Omron CX-Programmer project НовыйПроект (CX-Programmer 9.54)

# PLC НовыйПЛК1: CP1L-E EM

## Global symbols (name address type ; comment)
0.02 BOOL  ; EMG
0.08 BOOL  ; пустой латок
100.06 BOOL  ; лампа зеленой кнопки
C0000 BOOL  ; Счетчик шага ленты
C0001 BOOL  ; Счетчик часов
C0002 BOOL  ; Счетчик секунд
C0003 BOOL  ; Счетчик минут
C0004 BOOL  ; Счетчик счетчиков часов
C0005 BOOL  ; Счетчик ручного режима
C0006 BOOL  ; Счетчик аварий элеватора
C0007 BOOL  ; Счетчик аварий тарелки
C0008 BOOL  ; Счетчик нажатий грибка
C0009 BOOL  ; Счетчик реле безопасности
C0010 BOOL  ; счетсик секунд
C0011 BOOL  ; счетчик минут
C0012 BOOL  ; счтечик часов
C0013 BOOL  ; счетчик счетчика часов
C0014 BOOL  ; счетчик секунд
C0015 BOOL  ; счетчик минут
C0016 BOOL  ; счетчик часов
T0000 BOOL  ; Таймер задержки ленты
T0001 BOOL  ; лента не двигается
T0002 BOOL  ; Задержка включения ориентатора
T0005 BOOL  ; Задержка включения воздуха
T0006 BOOL  ; Задержка выключения ориентатора
T0010 BOOL  ; Наполнение тарелки
T0012 BOOL  ; лента не двигается
W0.03 BOOL  ; Ошибка связи с ПЧ
W0.04 BOOL  ; Связь с ПЧ ОК
W10.03 BOOL  ; Движение ленты с панели
W10.04 BOOL  ; Сброс
W1.01 BOOL  ; Ручная подача воздуха в трубу
W1.02 BOOL  ; Подача воздуха с панели
W1.09 BOOL  ; Сменился день
W2.01 BOOL  ; Общий сброс
W3.00 BOOL  ; сброс веремя работы
DayNew D600 UINT  ; Новый день
DayStar D602 UINT  ; День прошедший
LocAlarm D554 UINT
LocEMG D562 UINT
LocElev D558 UINT
LocManual D556 UINT
LocNotaus D564 UINT
LocTarelki D560 UINT
ResAlarm D504 UINT
ResEMG D512 UINT
ResElev D508 UINT
ResManual D506 UINT
ResNotaus D514 UINT
ResProst D500 UDINT  ; Простой после сброса
ResTarelki D510 UINT
ResWork D502 UDINT  ; Работа после сброса
Safety 0.00 BOOL  ; Реле безопасности
StatAlarm D464 UINT
StatEMG D468 UINT
StatElev D466 UINT
StatManual D465 UINT
StatNotaus D469 UINT
StatProst D460 UDINT  ; Глобальная статистика простоя
StatTarelki D467 UINT
StatWork D462 UDINT  ; Глобальная статистика работы
TimeSek A351 UINT
ghr INV002_Refresh_X31_
locProst D550 UDINT_BCD  ; время простоя локальное
locWork D552 UDINT_BCD  ; время работы локальное
time D400 UINT
Контроль_нового_дня Новый_день
Сброс_EMG Сброс2
Сброс_Ручного_режима Сброс2
Сброс_аварии_ленты Сброс2
Сброс_аварии_тарелки Сброс2
Сброс_аварии_терелки Сброс2
Сброс_времени_аварии Сброс2
Сброс_времени_работы Сброс
Сброс_реле_безопасности Сброс2
Смещение_EMG Сдвиг_данных2
Смещение_авари Сдвиг_данных2
Смещение_простоя сдвиг_данных
Смещение_работы сдвиг_данных
Смещение_реле_безопасности Сдвиг_данных2
Смещение_ручного Сдвиг_данных2
Смещение_тарелки Сдвиг_данных2
Смещение_элеватора Сдвиг_данных2
сброс_времени_простоя Сброс

## Program Ориентатор (cyclic task 0)
Local symbols
Air 100.00 BOOL  ; Подача воздуха
AirPipe 101.00 BOOL  ; Клапан воздуха в трубе
Alarm W0.02 BOOL  ; Сигнал ошибки
Alarm_Elevator W0.08 BOOL  ; Авария ленты
Alarm_Feeder W0.11 BOOL  ; Авария вращения тарелки
B1 0.04 BOOL  ; Заполнение тарелки
B2 0.03 BOOL  ; Уровень бункера
B3 0.06 BOOL  ; Шаг ленты
B4 0.05 BOOL  ; Вращение тарелки
B5 0.07 BOOL  ; Максимум лотка
DD434 INT
Flag W0.00 BOOL  ; Флаг старта
Freq D0 UINT  ; Задание частоты с панели
Green_Light 100.07 BOOL  ; Светофор зеленый
Manual W10.02 BOOL  ; Ручной режим
Power_Elevator 101.02 BOOL  ; Двигатель ленты
Power_Feeder W0.01 BOOL  ; Включение вращения тарелки
Red_Lamp 100.02 BOOL  ; Питание Реле
Red_Light 100.03 BOOL  ; Светофор красный
Reset W10.01 BOOL  ; Сброс
ResetSafety 100.01 BOOL  ; Сброс реле безопасности
Safety 0.00 BOOL  ; Реле безопасности
Sound 100.05 BOOL  ; Звук
Start W10.00 BOOL  ; Старт
Step D401 UINT_BCD  ; Количество шагов ленты
Timer1 D402 UINT_BCD  ; Задержка ленты
Timer2 D404 UINT_BCD  ; Задержка включения ориентатора
Timer3 D406 UINT_BCD  ; Задержка выключения ориентатора
Timer4 D408 UINT_BCD  ; Задержка подачи воздуха в трубе
Timer5 D410 UINT_BCD  ; Задержка отключения воздуха в трубе
Yellow_Light 100.04 BOOL  ; Светофор желтый
В431 CHANNEL
С13 INT

### Section Основная_программа

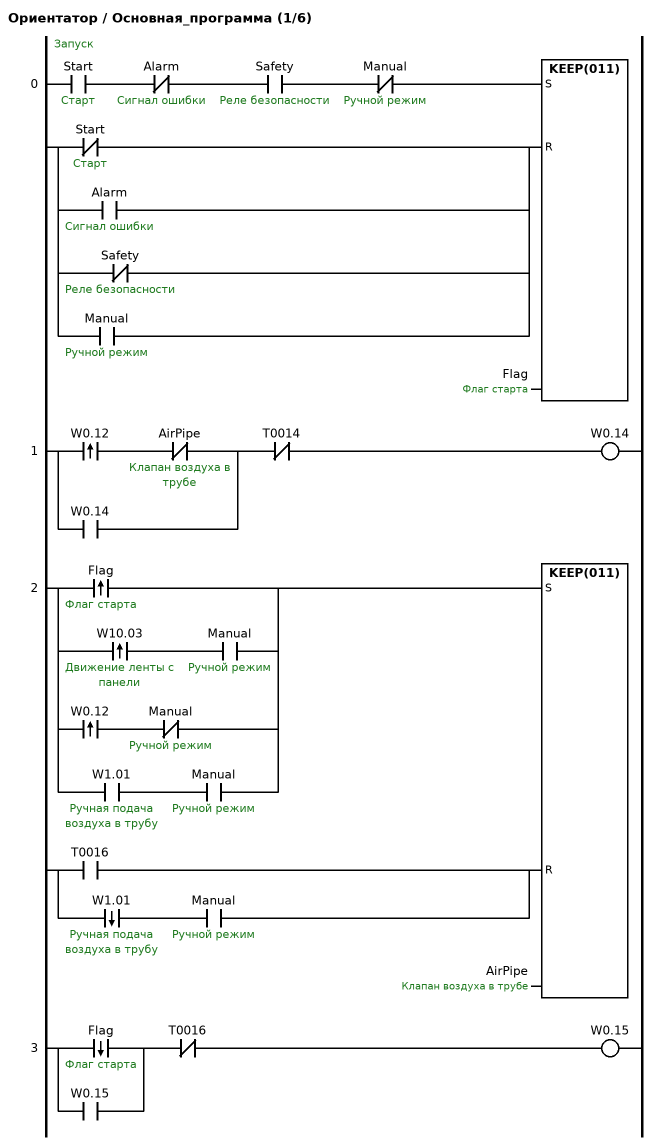
; rung 0: Запуск
LD Start  ; Старт
ANDNOT Alarm  ; Сигнал ошибки
AND Safety  ; Реле безопасности
ANDNOT Manual  ; Ручной режим
LDNOT Start  ; Старт
OR Alarm  ; Сигнал ошибки
ORNOT Safety  ; Реле безопасности
OR Manual  ; Ручной режим
KEEP(011) Flag  ; Флаг старта
; rung 1
@LD W0.12
ANDNOT AirPipe  ; Клапан воздуха в трубе
OR W0.14
ANDNOT T0014
OUT W0.14
; rung 2
@LD Flag  ; Флаг старта
@LD W10.03  ; Движение ленты с панели
AND Manual  ; Ручной режим
ORLD
@LD W0.12
ANDNOT Manual  ; Ручной режим
ORLD
LD W1.01  ; Ручная подача воздуха в трубу
AND Manual  ; Ручной режим
ORLD
LD T0016
%LD W1.01  ; Ручная подача воздуха в трубу
AND Manual  ; Ручной режим
ORLD
KEEP(011) AirPipe  ; Клапан воздуха в трубе
; rung 3
%LD Flag  ; Флаг старта
OR W0.15
ANDNOT T0016
OUT W0.15

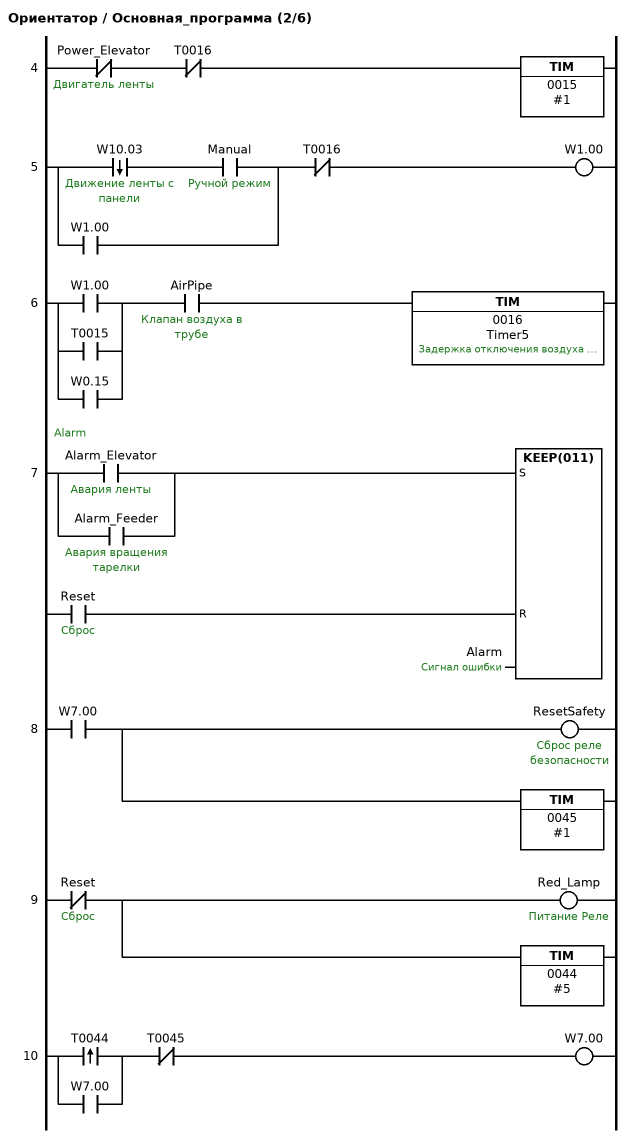
; rung 4
LDNOT Power_Elevator  ; Двигатель ленты
ANDNOT T0016
TIM 0015 #1
; rung 5
%LD W10.03  ; Движение ленты с панели
AND Manual  ; Ручной режим
OR W1.00
ANDNOT T0016
OUT W1.00
; rung 6
LD W1.00
OR T0015
OR W0.15
AND AirPipe  ; Клапан воздуха в трубе
TIM 0016 Timer5  ; Задержка отключения воздуха в трубе
; rung 7: Alarm
LD Alarm_Elevator  ; Авария ленты
OR Alarm_Feeder  ; Авария вращения тарелки
LD Reset  ; Сброс
KEEP(011) Alarm  ; Сигнал ошибки
; rung 8
LD W7.00
OUT ResetSafety  ; Сброс реле безопасности
TIM 0045 #1
; rung 9
LDNOT Reset  ; Сброс
OUT Red_Lamp  ; Питание Реле
TIM 0044 #5
; rung 10
@LD T0044
OR W7.00
ANDNOT T0045
OUT W7.00

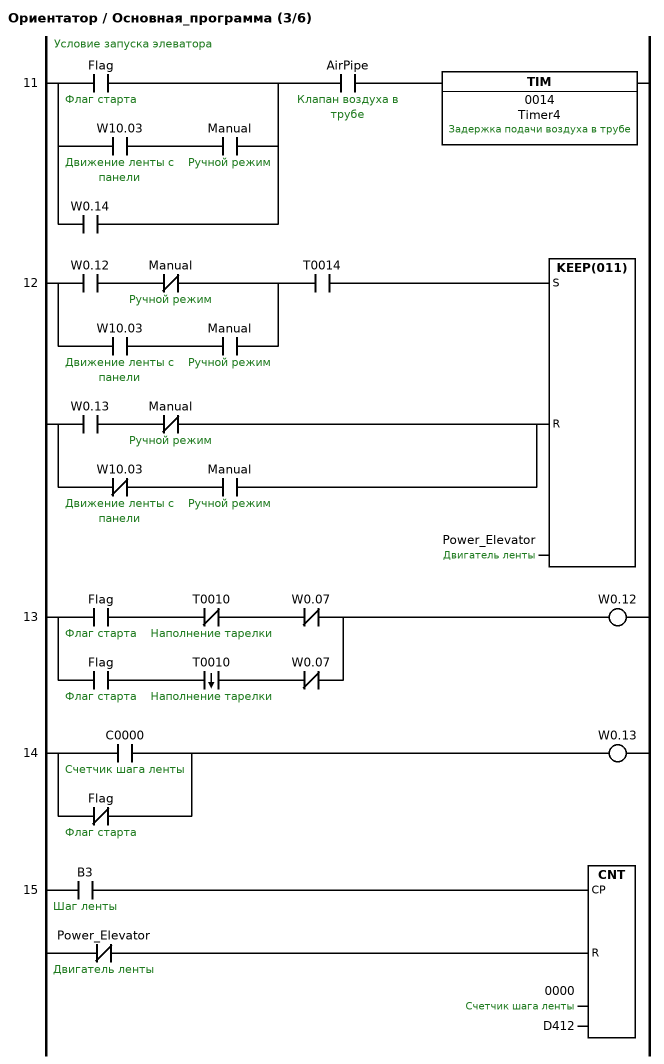
; rung 11: Условие запуска элеватора
LD Flag  ; Флаг старта
LD W10.03  ; Движение ленты с панели
AND Manual  ; Ручной режим
ORLD
OR W0.14
AND AirPipe  ; Клапан воздуха в трубе
TIM 0014 Timer4  ; Задержка подачи воздуха в трубе
; rung 12
LD W0.12
ANDNOT Manual  ; Ручной режим
LD W10.03  ; Движение ленты с панели
AND Manual  ; Ручной режим
ORLD
AND T0014
LD W0.13
ANDNOT Manual  ; Ручной режим
LDNOT W10.03  ; Движение ленты с панели
AND Manual  ; Ручной режим
ORLD
KEEP(011) Power_Elevator  ; Двигатель ленты
; rung 13
LD Flag  ; Флаг старта
ANDNOT T0010  ; Наполнение тарелки
ANDNOT W0.07
LD Flag  ; Флаг старта
%AND T0010  ; Наполнение тарелки
ANDNOT W0.07
ORLD
OUT W0.12
; rung 14
LD C0000  ; Счетчик шага ленты
ORNOT Flag  ; Флаг старта
OUT W0.13
; rung 15
LD B3  ; Шаг ленты
LDNOT Power_Elevator  ; Двигатель ленты
CNT 0000 D412  ; Счетчик шага ленты

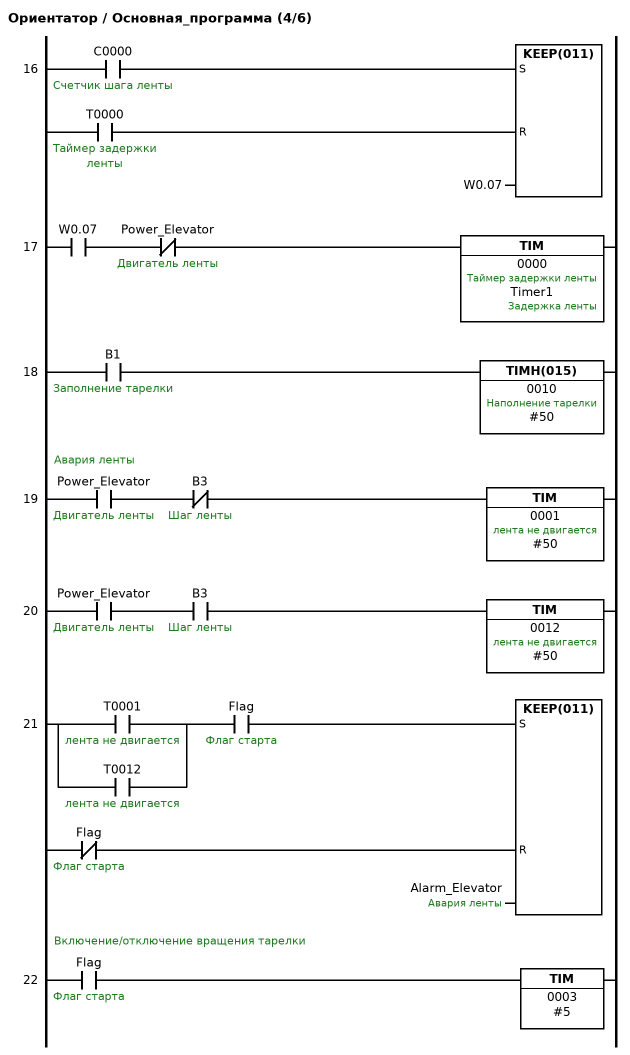
; rung 16
LD C0000  ; Счетчик шага ленты
LD T0000  ; Таймер задержки ленты
KEEP(011) W0.07
; rung 17
LD W0.07
ANDNOT Power_Elevator  ; Двигатель ленты
TIM 0000 Timer1  ; Задержка ленты, Таймер задержки ленты
; rung 18
LD B1  ; Заполнение тарелки
TIMH(015) 0010 #50  ; Наполнение тарелки
; rung 19: Авария ленты
LD Power_Elevator  ; Двигатель ленты
ANDNOT B3  ; Шаг ленты
TIM 0001 #50  ; лента не двигается
; rung 20
LD Power_Elevator  ; Двигатель ленты
AND B3  ; Шаг ленты
TIM 0012 #50  ; лента не двигается
; rung 21
LD T0001  ; лента не двигается
OR T0012  ; лента не двигается
AND Flag  ; Флаг старта
LDNOT Flag  ; Флаг старта
KEEP(011) Alarm_Elevator  ; Авария ленты
; rung 22: Включение/отключение вращения тарелки
LD Flag  ; Флаг старта
TIM 0003 #5

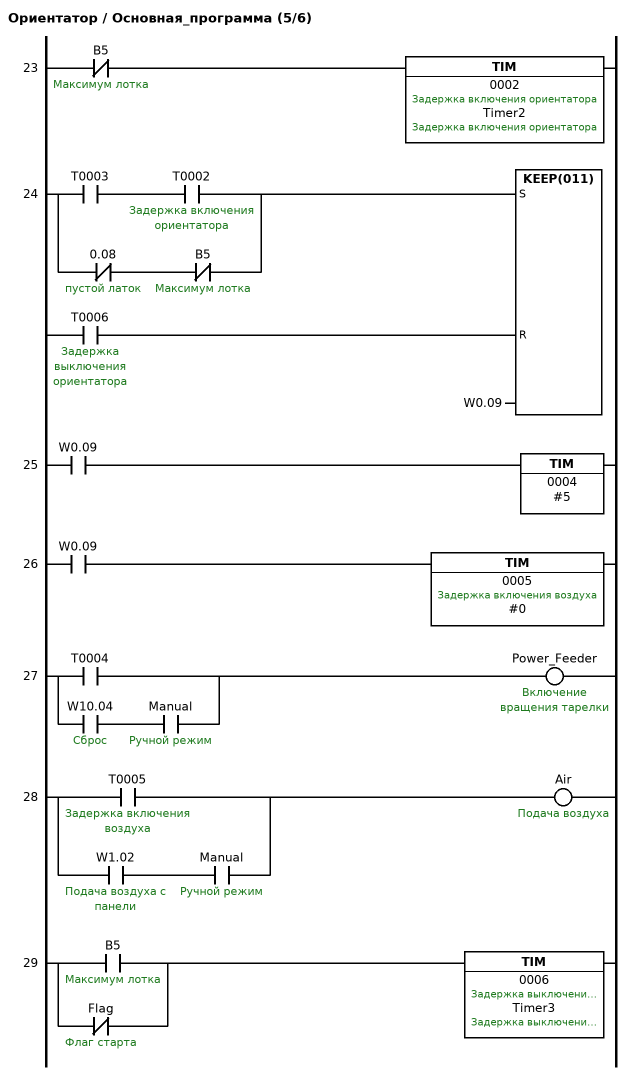
; rung 23
LDNOT B5  ; Максимум лотка
TIM 0002 Timer2  ; Задержка включения ориентатора
; rung 24
LD T0003
AND T0002  ; Задержка включения ориентатора
LDNOT 0.08  ; пустой латок
ANDNOT B5  ; Максимум лотка
ORLD
LD T0006  ; Задержка выключения ориентатора
KEEP(011) W0.09
; rung 25
LD W0.09
TIM 0004 #5
; rung 26
LD W0.09
TIM 0005 #0  ; Задержка включения воздуха
; rung 27
LD T0004
LD W10.04  ; Сброс
AND Manual  ; Ручной режим
ORLD
OUT Power_Feeder  ; Включение вращения тарелки
; rung 28
LD T0005  ; Задержка включения воздуха
LD W1.02  ; Подача воздуха с панели
AND Manual  ; Ручной режим
ORLD
OUT Air  ; Подача воздуха
; rung 29
LD B5  ; Максимум лотка
ORNOT Flag  ; Флаг старта
TIM 0006 Timer3  ; Задержка выключения ориентатора

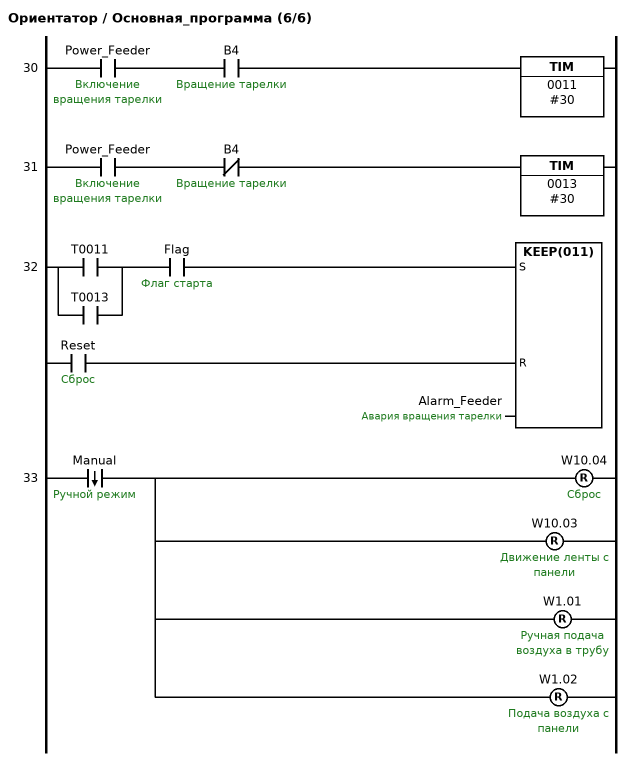
; rung 30
LD Power_Feeder  ; Включение вращения тарелки
AND B4  ; Вращение тарелки
TIM 0011 #30
; rung 31
LD Power_Feeder  ; Включение вращения тарелки
ANDNOT B4  ; Вращение тарелки
TIM 0013 #30
; rung 32
LD T0011
OR T0013
AND Flag  ; Флаг старта
LD Reset  ; Сброс
KEEP(011) Alarm_Feeder  ; Авария вращения тарелки
; rung 33
%LD Manual  ; Ручной режим
RSET W10.04  ; Сброс
RSET W10.03  ; Движение ленты с панели
RSET W1.01  ; Ручная подача воздуха в трубу
RSET W1.02  ; Подача воздуха с панели

### Section Частотник

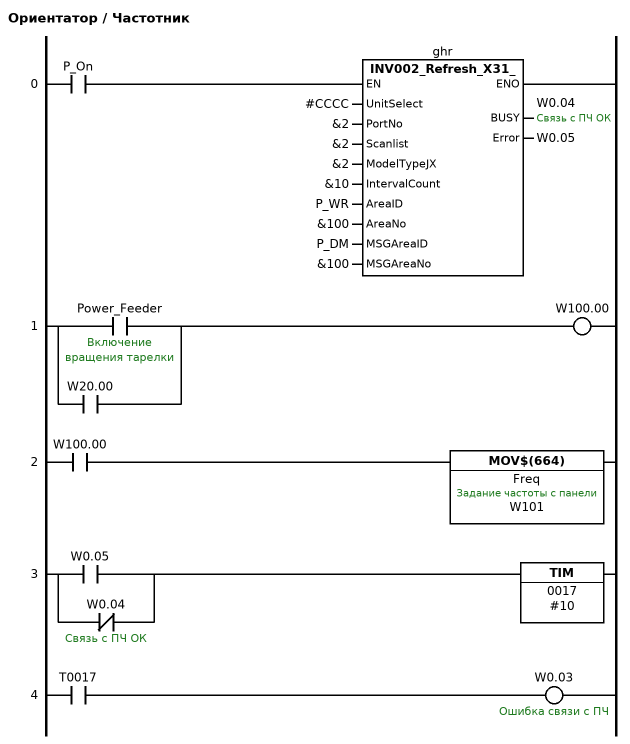
; rung 0
LD P_On
CALL ghr : INV002_Refresh_X31_ (UnitSelect := #CCCC, PortNo := &2, Scanlist := &2, ModelTypeJX := &2, IntervalCount := &10, AreaID := P_WR, AreaNo := &100, MSGAreaID := P_DM, MSGAreaNo := &100, BUSY => W0.04, Error => W0.05)  ; Связь с ПЧ ОК
; rung 1
LD Power_Feeder  ; Включение вращения тарелки
OR W20.00
OUT W100.00
; rung 2
LD W100.00
MOV$(664) Freq W101  ; Задание частоты с панели
; rung 3
LD W0.05
ORNOT W0.04  ; Связь с ПЧ ОК
TIM 0017 #10
; rung 4
LD T0017
OUT W0.03  ; Ошибка связи с ПЧ

### Section Индикация

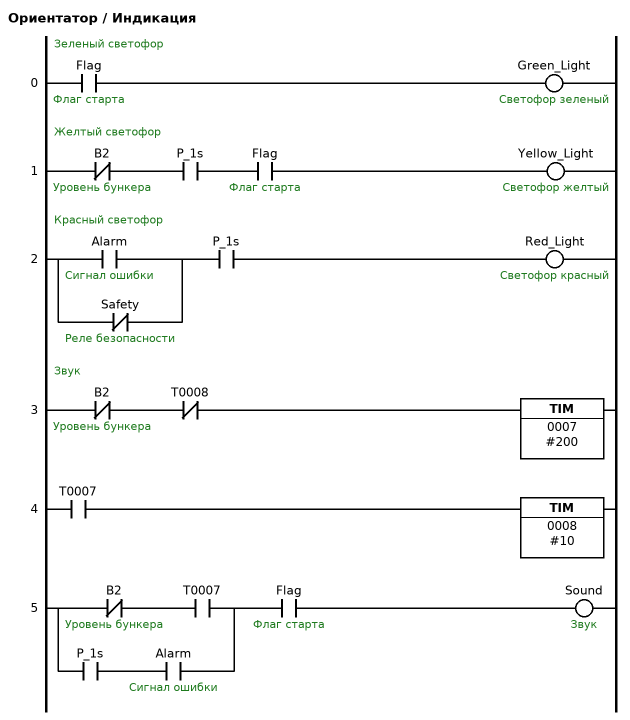
; rung 0: Зеленый светофор
LD Flag  ; Флаг старта
OUT Green_Light  ; Светофор зеленый
; rung 1: Желтый светофор
LDNOT B2  ; Уровень бункера
AND P_1s
AND Flag  ; Флаг старта
OUT Yellow_Light  ; Светофор желтый
; rung 2: Красный светофор
LD Alarm  ; Сигнал ошибки
ORNOT Safety  ; Реле безопасности
AND P_1s
OUT Red_Light  ; Светофор красный
; rung 3: Звук
LDNOT B2  ; Уровень бункера
ANDNOT T0008
TIM 0007 #200
; rung 4
LD T0007
TIM 0008 #10
; rung 5
LDNOT B2  ; Уровень бункера
AND T0007
LD P_1s
AND Alarm  ; Сигнал ошибки
ORLD
AND Flag  ; Флаг старта
OUT Sound  ; Звук

### Section End
; rung 0
END(001)

## Program статистика (cyclic task 1)
Local symbols
Alarm W0.02 BOOL  ; Сигнал ошибки
AlarmDay1 D628 UINT
AlarmDay2 D629 UINT
AlarmDay3 D630 UINT
Alarm_Elevator W0.08 BOOL  ; Авария ленты
Alarm_Feeder W0.11 BOOL  ; Авария вращения тарелки
Day1 D613 UINT
Day2 D616 UINT
Day3 D619 UINT
DayNew D600 UINT
DayStar D602 UINT
EMGDay1 D644 UINT
EMGDay2 D645 UINT
EMGDay3 D646 UINT
ElevDay1 D636 UINT
ElevDay2 D637 UINT
ElevDay3 D638 UINT
Flag W0.00 BOOL  ; Флаг старта
LocProst D550 UDINT
LocWork D552 UDINT
Manual W10.02 BOOL  ; Ручной режим
ManualDay1 D632 UINT
ManualDay2 D633 UINT
ManualDay3 D634 UINT
Mon1 D614 UINT
Mon2 D617 UINT
Mon3 D620 UINT
MonNew D601 UINT
MonStar D603 UINT
NotausDay1 D648 UINT
NotausDay2 D649 UINT
NotausDay3 D650 UINT
ProstDay1 D612 UINT  ; Простой 1 день
ProstDay2 D615 UINT  ; Простой 2 день
ProstDay3 D618 UINT  ; Простой 3 день
TarelkaDay1 D640 UINT
TarelkaDay2 D641 UINT
TarelkaDay3 D642 UINT
TochOtschAlarm D626 UINT
TochOtschEMG D643 UINT
TochOtschElev D635 UINT
TochOtschManual D631 UINT
TochOtschNotaus D647 UINT
TochOtschProst D610 UDINT
TochOtschTarelki D639 UINT
TochOtschWork D621 UDINT
WorkDay1 D623 UINT  ; работа 1 дня
WorkDay2 D624 UINT  ; Работа 2 дня
WorkDay3 D625 UINT  ; Работа 3 дня

### Section Сбор_статистики

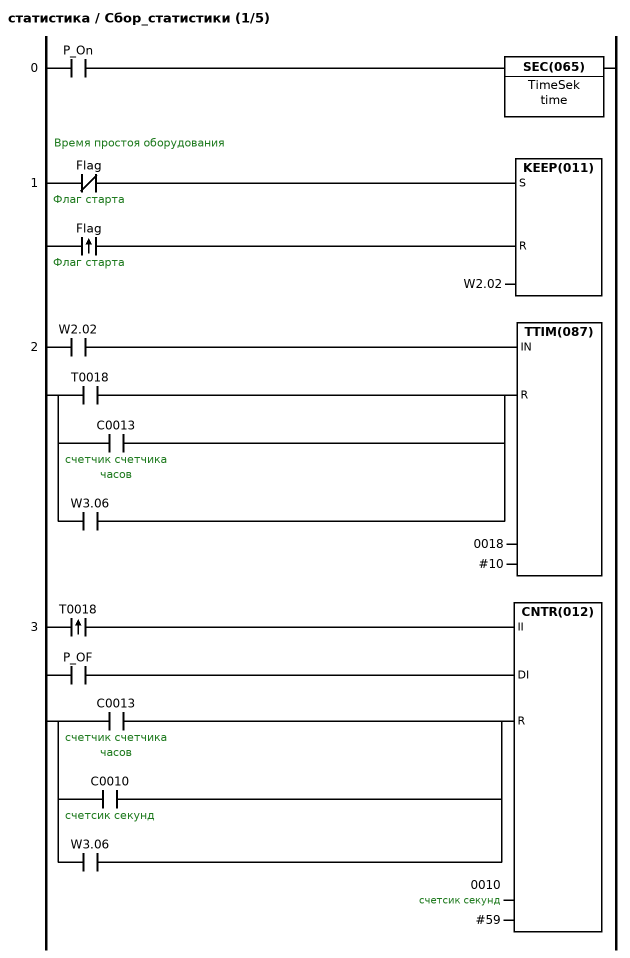
; rung 0
LD P_On
SEC(065) TimeSek time
; rung 1: Время простоя оборудования
LDNOT Flag  ; Флаг старта
@LD Flag  ; Флаг старта
KEEP(011) W2.02
; rung 2
LD W2.02
LD T0018
OR C0013  ; счетчик счетчика часов
OR W3.06
TTIM(087) 0018 #10
; rung 3
@LD T0018
LD P_OF
LD C0013  ; счетчик счетчика часов
OR C0010  ; счетсик секунд
OR W3.06
CNTR(012) 0010 #59  ; счетсик секунд

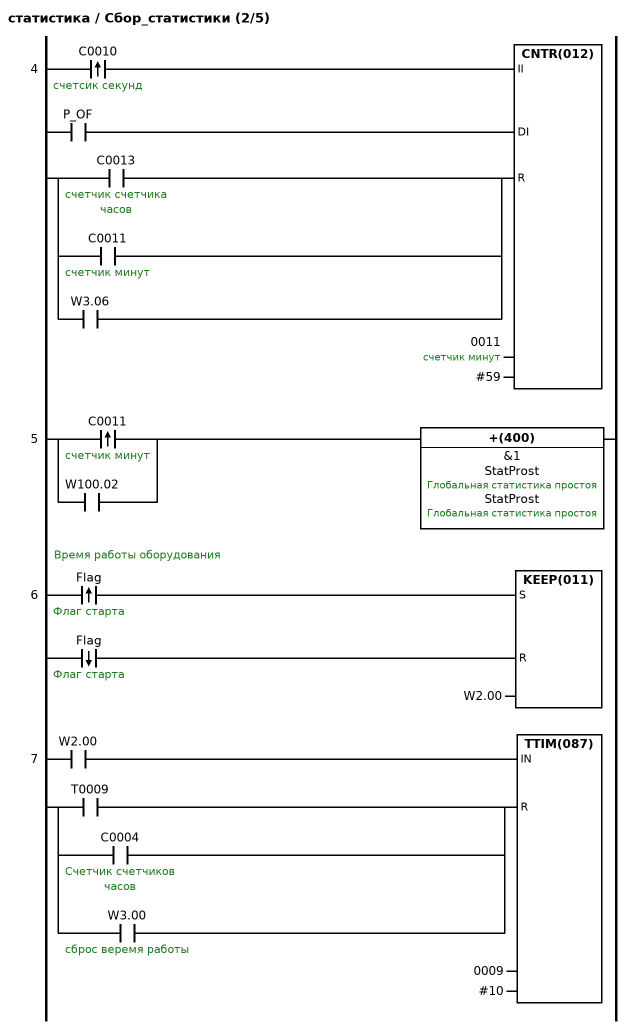
; rung 4
@LD C0010  ; счетсик секунд
LD P_OF
LD C0013  ; счетчик счетчика часов
OR C0011  ; счетчик минут
OR W3.06
CNTR(012) 0011 #59  ; счетчик минут
; rung 5
@LD C0011  ; счетчик минут
OR W100.02
+(400) &1 StatProst StatProst  ; Глобальная статистика простоя
; rung 6: Время работы оборудования
@LD Flag  ; Флаг старта
%LD Flag  ; Флаг старта
KEEP(011) W2.00
; rung 7
LD W2.00
LD T0009
OR C0004  ; Счетчик счетчиков часов
OR W3.00  ; сброс веремя работы
TTIM(087) 0009 #10

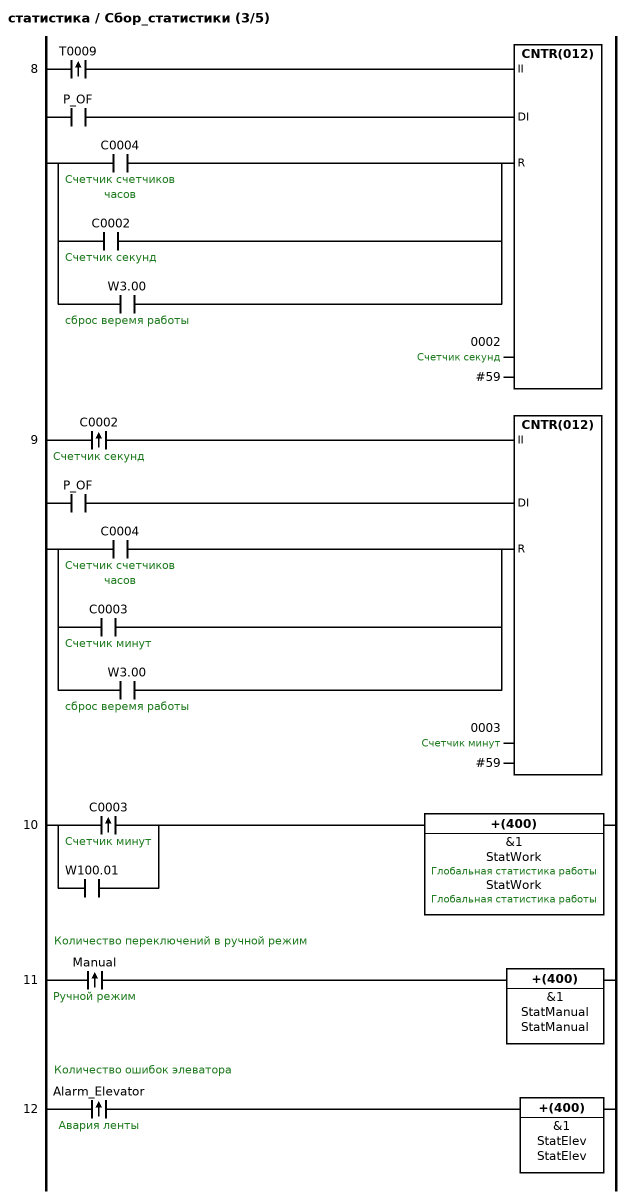
; rung 8
@LD T0009
LD P_OF
LD C0004  ; Счетчик счетчиков часов
OR C0002  ; Счетчик секунд
OR W3.00  ; сброс веремя работы
CNTR(012) 0002 #59  ; Счетчик секунд
; rung 9
@LD C0002  ; Счетчик секунд
LD P_OF
LD C0004  ; Счетчик счетчиков часов
OR C0003  ; Счетчик минут
OR W3.00  ; сброс веремя работы
CNTR(012) 0003 #59  ; Счетчик минут
; rung 10
@LD C0003  ; Счетчик минут
OR W100.01
+(400) &1 StatWork StatWork  ; Глобальная статистика работы
; rung 11: Количество переключений в ручной режим
@LD Manual  ; Ручной режим
+(400) &1 StatManual StatManual
; rung 12: Количество ошибок элеватора
@LD Alarm_Elevator  ; Авария ленты
+(400) &1 StatElev StatElev

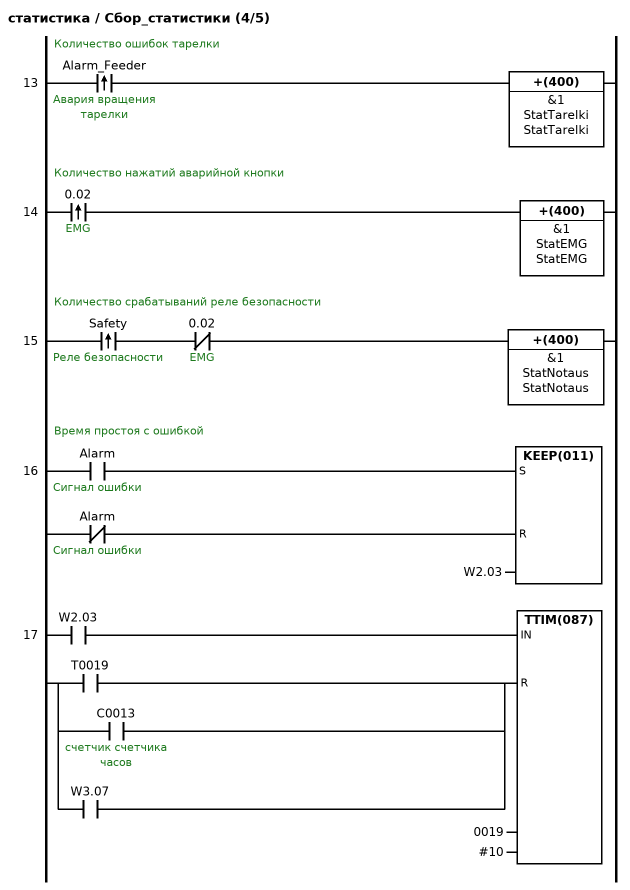
; rung 13: Количество ошибок тарелки
@LD Alarm_Feeder  ; Авария вращения тарелки
+(400) &1 StatTarelki StatTarelki
; rung 14: Количество нажатий аварийной кнопки
@LD 0.02  ; EMG
+(400) &1 StatEMG StatEMG
; rung 15: Количество срабатываний реле безопасности
@LD Safety  ; Реле безопасности
ANDNOT 0.02  ; EMG
+(400) &1 StatNotaus StatNotaus
; rung 16: Время простоя с ошибкой
LD Alarm  ; Сигнал ошибки
LDNOT Alarm  ; Сигнал ошибки
KEEP(011) W2.03
; rung 17
LD W2.03
LD T0019
OR C0013  ; счетчик счетчика часов
OR W3.07
TTIM(087) 0019 #10

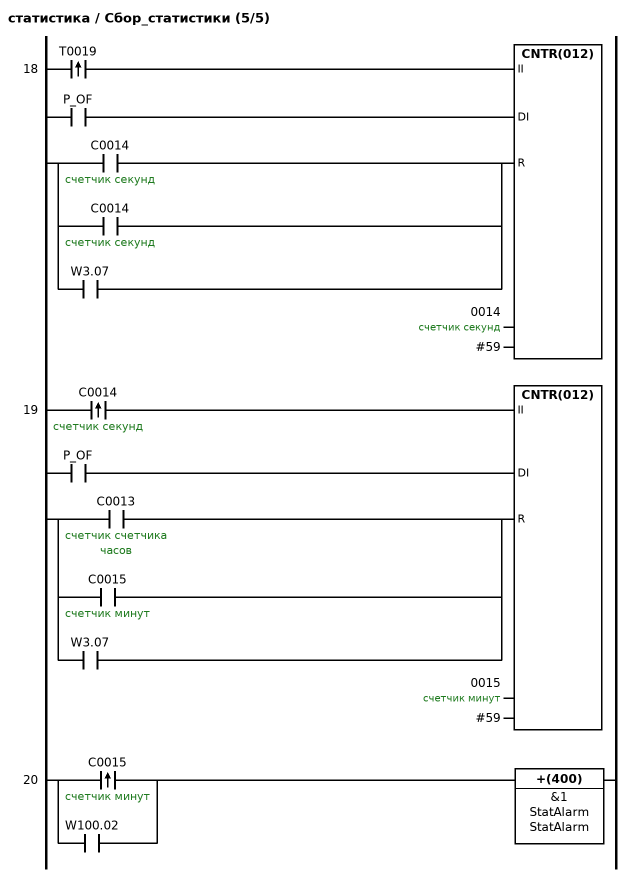
; rung 18
@LD T0019
LD P_OF
LD C0014  ; счетчик секунд
OR C0014  ; счетчик секунд
OR W3.07
CNTR(012) 0014 #59  ; счетчик секунд
; rung 19
@LD C0014  ; счетчик секунд
LD P_OF
LD C0013  ; счетчик счетчика часов
OR C0015  ; счетчик минут
OR W3.07
CNTR(012) 0015 #59  ; счетчик минут
; rung 20
@LD C0015  ; счетчик минут
OR W100.02
+(400) &1 StatAlarm StatAlarm

### Section расчет_статистики

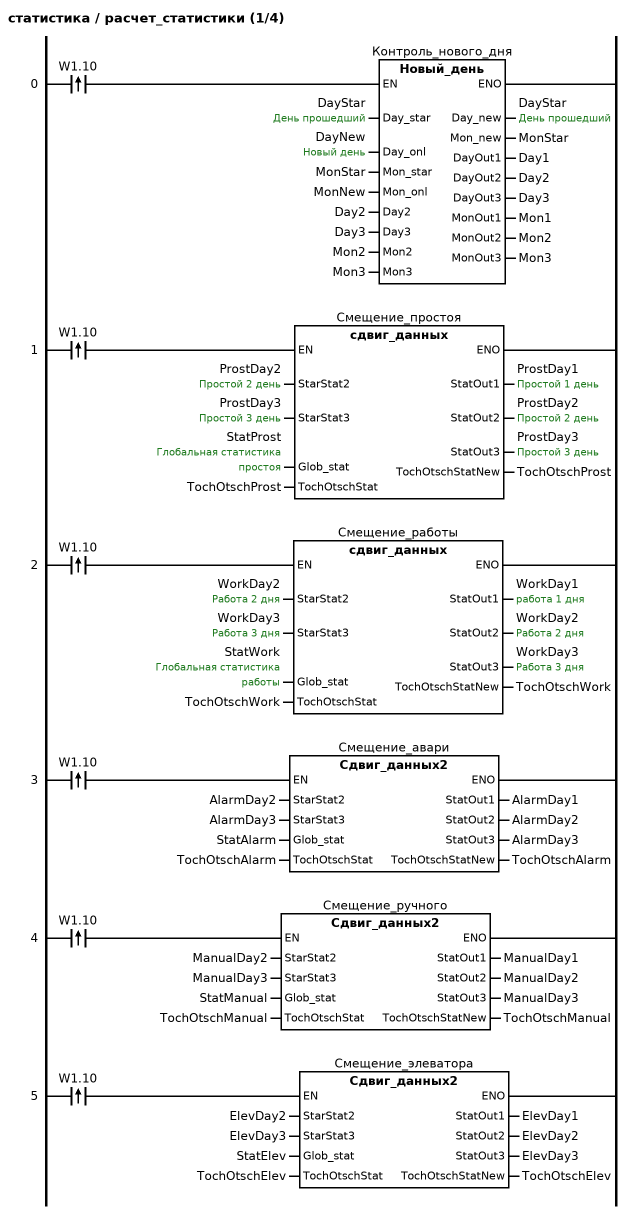
; rung 0
@LD W1.10
CALL Контроль_нового_дня : Новый_день (Day_star := DayStar, Day_onl := DayNew, Mon_star := MonStar, Mon_onl := MonNew, Day2 := Day2, Day3 := Day3, Mon2 := Mon2, Mon3 := Mon3, Day_new => DayStar, Mon_new => MonStar, DayOut1 => Day1, DayOut2 => Day2, DayOut3 => Day3, MonOut1 => Mon1, MonOut2 => Mon2, MonOut3 => Mon3)  ; День прошедший, Новый день
; rung 1
@LD W1.10
CALL Смещение_простоя : сдвиг_данных (StarStat2 := ProstDay2, StarStat3 := ProstDay3, Glob_stat := StatProst, TochOtschStat := TochOtschProst, StatOut1 => ProstDay1, StatOut2 => ProstDay2, StatOut3 => ProstDay3, TochOtschStatNew => TochOtschProst)  ; Простой 2 день, Простой 3 день, Глобальная статистика простоя, Простой 1 день
; rung 2
@LD W1.10
CALL Смещение_работы : сдвиг_данных (StarStat2 := WorkDay2, StarStat3 := WorkDay3, Glob_stat := StatWork, TochOtschStat := TochOtschWork, StatOut1 => WorkDay1, StatOut2 => WorkDay2, StatOut3 => WorkDay3, TochOtschStatNew => TochOtschWork)  ; Работа 2 дня, Работа 3 дня, Глобальная статистика работы, работа 1 дня
; rung 3
@LD W1.10
CALL Смещение_авари : Сдвиг_данных2 (StarStat2 := AlarmDay2, StarStat3 := AlarmDay3, Glob_stat := StatAlarm, TochOtschStat := TochOtschAlarm, StatOut1 => AlarmDay1, StatOut2 => AlarmDay2, StatOut3 => AlarmDay3, TochOtschStatNew => TochOtschAlarm)
; rung 4
@LD W1.10
CALL Смещение_ручного : Сдвиг_данных2 (StarStat2 := ManualDay2, StarStat3 := ManualDay3, Glob_stat := StatManual, TochOtschStat := TochOtschManual, StatOut1 => ManualDay1, StatOut2 => ManualDay2, StatOut3 => ManualDay3, TochOtschStatNew => TochOtschManual)
; rung 5
@LD W1.10
CALL Смещение_элеватора : Сдвиг_данных2 (StarStat2 := ElevDay2, StarStat3 := ElevDay3, Glob_stat := StatElev, TochOtschStat := TochOtschElev, StatOut1 => ElevDay1, StatOut2 => ElevDay2, StatOut3 => ElevDay3, TochOtschStatNew => TochOtschElev)

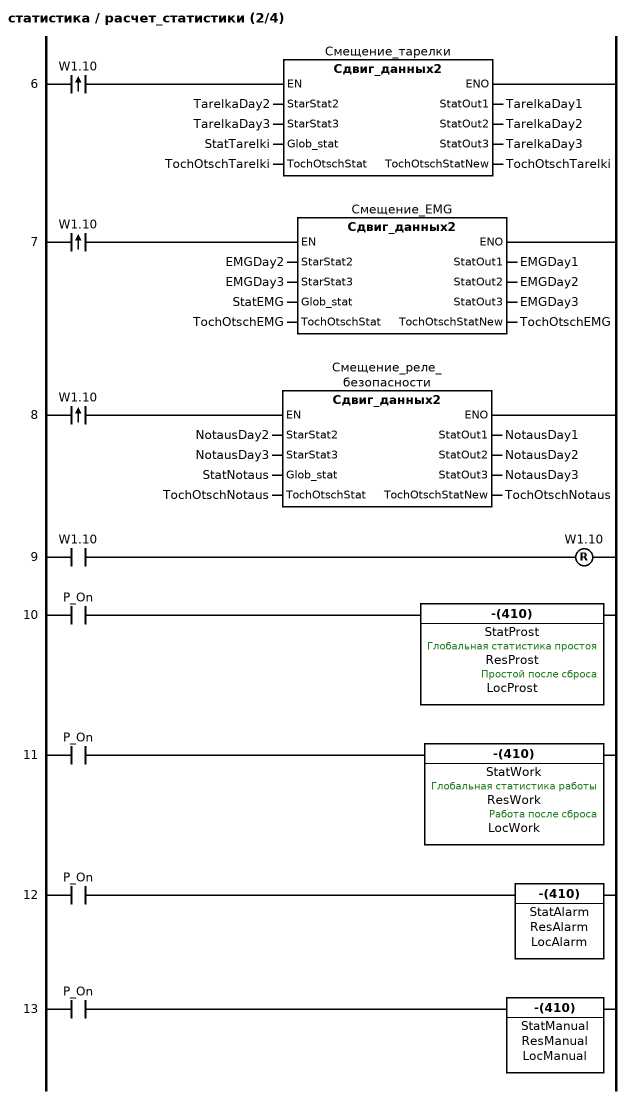
; rung 6
@LD W1.10
CALL Смещение_тарелки : Сдвиг_данных2 (StarStat2 := TarelkaDay2, StarStat3 := TarelkaDay3, Glob_stat := StatTarelki, TochOtschStat := TochOtschTarelki, StatOut1 => TarelkaDay1, StatOut2 => TarelkaDay2, StatOut3 => TarelkaDay3, TochOtschStatNew => TochOtschTarelki)
; rung 7
@LD W1.10
CALL Смещение_EMG : Сдвиг_данных2 (StarStat2 := EMGDay2, StarStat3 := EMGDay3, Glob_stat := StatEMG, TochOtschStat := TochOtschEMG, StatOut1 => EMGDay1, StatOut2 => EMGDay2, StatOut3 => EMGDay3, TochOtschStatNew => TochOtschEMG)
; rung 8
@LD W1.10
CALL Смещение_реле_безопасности : Сдвиг_данных2 (StarStat2 := NotausDay2, StarStat3 := NotausDay3, Glob_stat := StatNotaus, TochOtschStat := TochOtschNotaus, StatOut1 => NotausDay1, StatOut2 => NotausDay2, StatOut3 => NotausDay3, TochOtschStatNew => TochOtschNotaus)
; rung 9
LD W1.10
RSET W1.10
; rung 10
LD P_On
-(410) StatProst ResProst LocProst  ; Глобальная статистика простоя, Простой после сброса
; rung 11
LD P_On
-(410) StatWork ResWork LocWork  ; Глобальная статистика работы, Работа после сброса
; rung 12
LD P_On
-(410) StatAlarm ResAlarm LocAlarm
; rung 13
LD P_On
-(410) StatManual ResManual LocManual

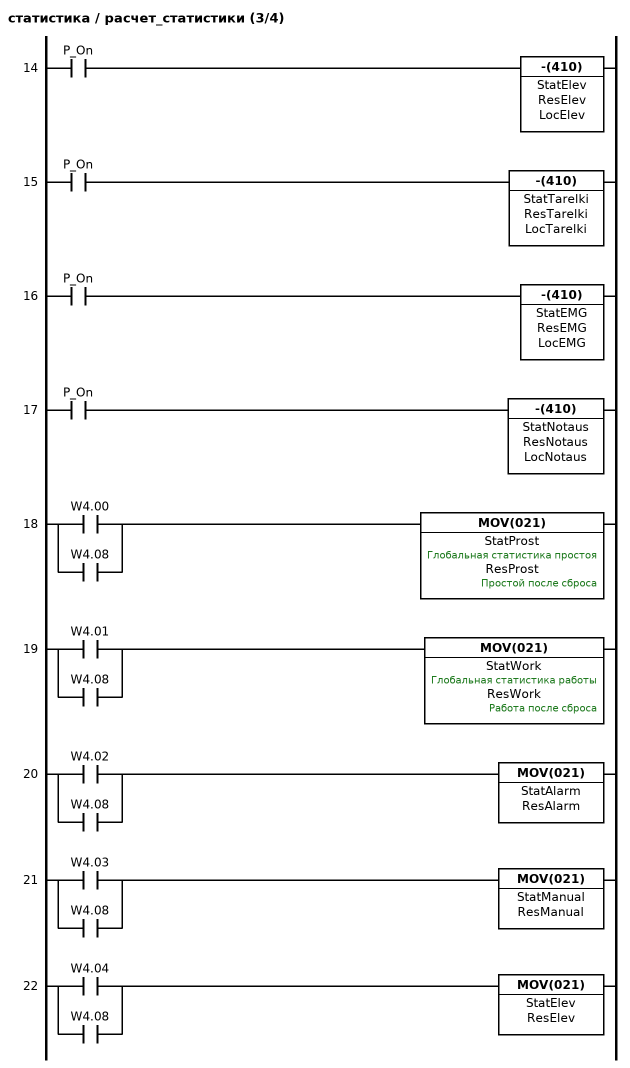
; rung 14
LD P_On
-(410) StatElev ResElev LocElev
; rung 15
LD P_On
-(410) StatTarelki ResTarelki LocTarelki
; rung 16
LD P_On
-(410) StatEMG ResEMG LocEMG
; rung 17
LD P_On
-(410) StatNotaus ResNotaus LocNotaus
; rung 18
LD W4.00
OR W4.08
MOV(021) StatProst ResProst  ; Глобальная статистика простоя, Простой после сброса
; rung 19
LD W4.01
OR W4.08
MOV(021) StatWork ResWork  ; Глобальная статистика работы, Работа после сброса
; rung 20
LD W4.02
OR W4.08
MOV(021) StatAlarm ResAlarm
; rung 21
LD W4.03
OR W4.08
MOV(021) StatManual ResManual
; rung 22
LD W4.04
OR W4.08
MOV(021) StatElev ResElev

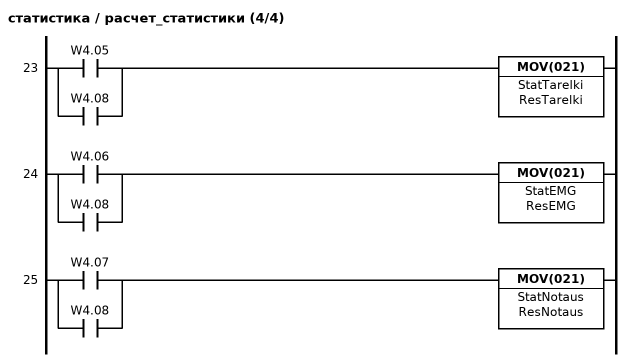
; rung 23
LD W4.05
OR W4.08
MOV(021) StatTarelki ResTarelki
; rung 24
LD W4.06
OR W4.08
MOV(021) StatEMG ResEMG
; rung 25
LD W4.07
OR W4.08
MOV(021) StatNotaus ResNotaus

### Section Сброс_статистики

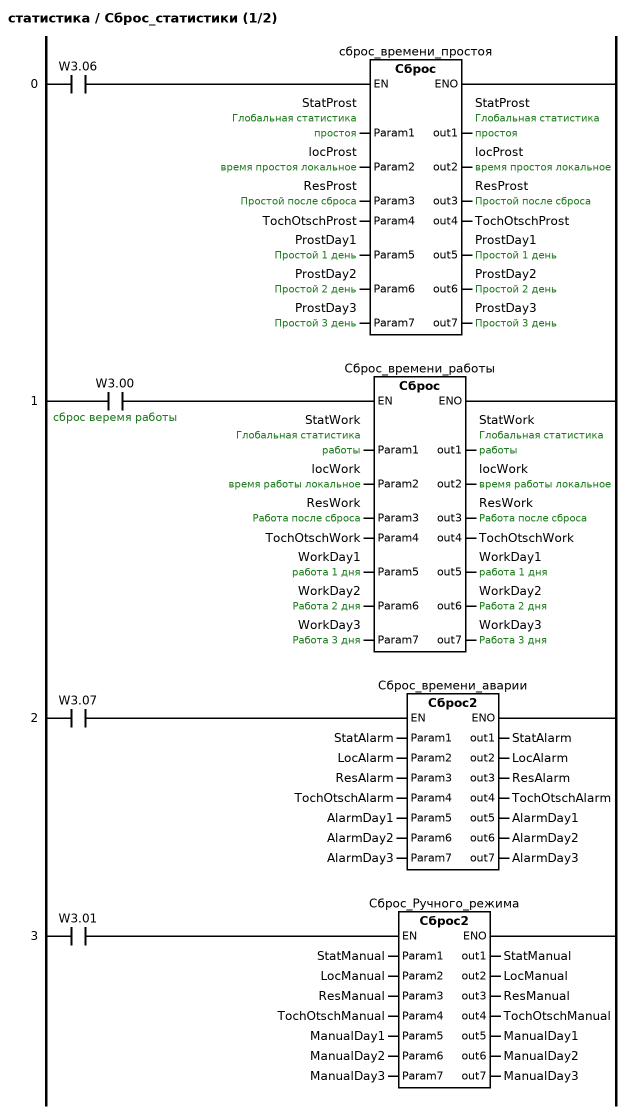
; rung 0
LD W3.06
CALL сброс_времени_простоя : Сброс (Param1 := StatProst, Param2 := locProst, Param3 := ResProst, Param4 := TochOtschProst, Param5 := ProstDay1, Param6 := ProstDay2, Param7 := ProstDay3, out1 => StatProst, out2 => locProst, out3 => ResProst, out4 => TochOtschProst, out5 => ProstDay1, out6 => ProstDay2, out7 => ProstDay3)  ; Глобальная статистика простоя, время простоя локальное, Простой после сброса, Простой 1 день, Простой 2 день, Простой 3 день
; rung 1
LD W3.00  ; сброс веремя работы
CALL Сброс_времени_работы : Сброс (Param1 := StatWork, Param2 := locWork, Param3 := ResWork, Param4 := TochOtschWork, Param5 := WorkDay1, Param6 := WorkDay2, Param7 := WorkDay3, out1 => StatWork, out2 => locWork, out3 => ResWork, out4 => TochOtschWork, out5 => WorkDay1, out6 => WorkDay2, out7 => WorkDay3)  ; Глобальная статистика работы, время работы локальное, Работа после сброса, работа 1 дня, Работа 2 дня, Работа 3 дня
; rung 2
LD W3.07
CALL Сброс_времени_аварии : Сброс2 (Param1 := StatAlarm, Param2 := LocAlarm, Param3 := ResAlarm, Param4 := TochOtschAlarm, Param5 := AlarmDay1, Param6 := AlarmDay2, Param7 := AlarmDay3, out1 => StatAlarm, out2 => LocAlarm, out3 => ResAlarm, out4 => TochOtschAlarm, out5 => AlarmDay1, out6 => AlarmDay2, out7 => AlarmDay3)
; rung 3
LD W3.01
CALL Сброс_Ручного_режима : Сброс2 (Param1 := StatManual, Param2 := LocManual, Param3 := ResManual, Param4 := TochOtschManual, Param5 := ManualDay1, Param6 := ManualDay2, Param7 := ManualDay3, out1 => StatManual, out2 => LocManual, out3 => ResManual, out4 => TochOtschManual, out5 => ManualDay1, out6 => ManualDay2, out7 => ManualDay3)

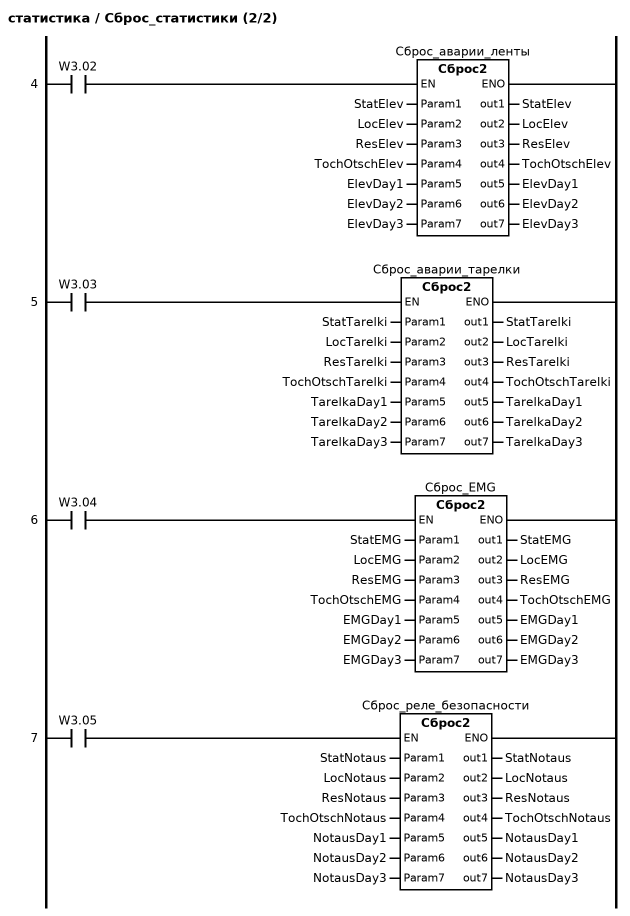
; rung 4
LD W3.02
CALL Сброс_аварии_ленты : Сброс2 (Param1 := StatElev, Param2 := LocElev, Param3 := ResElev, Param4 := TochOtschElev, Param5 := ElevDay1, Param6 := ElevDay2, Param7 := ElevDay3, out1 => StatElev, out2 => LocElev, out3 => ResElev, out4 => TochOtschElev, out5 => ElevDay1, out6 => ElevDay2, out7 => ElevDay3)
; rung 5
LD W3.03
CALL Сброс_аварии_тарелки : Сброс2 (Param1 := StatTarelki, Param2 := LocTarelki, Param3 := ResTarelki, Param4 := TochOtschTarelki, Param5 := TarelkaDay1, Param6 := TarelkaDay2, Param7 := TarelkaDay3, out1 => StatTarelki, out2 => LocTarelki, out3 => ResTarelki, out4 => TochOtschTarelki, out5 => TarelkaDay1, out6 => TarelkaDay2, out7 => TarelkaDay3)
; rung 6
LD W3.04
CALL Сброс_EMG : Сброс2 (Param1 := StatEMG, Param2 := LocEMG, Param3 := ResEMG, Param4 := TochOtschEMG, Param5 := EMGDay1, Param6 := EMGDay2, Param7 := EMGDay3, out1 => StatEMG, out2 => LocEMG, out3 => ResEMG, out4 => TochOtschEMG, out5 => EMGDay1, out6 => EMGDay2, out7 => EMGDay3)
; rung 7
LD W3.05
CALL Сброс_реле_безопасности : Сброс2 (Param1 := StatNotaus, Param2 := LocNotaus, Param3 := ResNotaus, Param4 := TochOtschNotaus, Param5 := NotausDay1, Param6 := NotausDay2, Param7 := NotausDay3, out1 => StatNotaus, out2 => LocNotaus, out3 => ResNotaus, out4 => TochOtschNotaus, out5 => NotausDay1, out6 => NotausDay2, out7 => NotausDay3)

### Section END
; rung 0
END(001)

## Function block INV002_Refresh_X31_
; <Status Refresh>Refreshes inverter status.
VAR_INPUT
  UnitSelect : INT;  (* Specify the connetcted Unit SCB=#BBBB_SCU=&0to&15 *)
  PortNo : INT := 1;  (* Serial port No. &0to&2 *)
  Scanlist : DWORD;  (* Scanlist *)
  ModelTypeJX : DWORD;  (* JX/MX or MX2/RX Classification for older Inverter types also this Bit has to be set, like scanlist *)
  IntervalCount : UINT;  (* Interval *)
  AreaID : WORD;  (* Using Area Classification *)
  AreaNo : INT;  (* Using Area Number *)
  MSGAreaID : WORD;  (* Message Area Classification *)
  MSGAreaNo : INT;  (* Message Area Number *)
END_VAR
VAR_OUTPUT
  BUSY : BOOL;  (* Processing Flag 0:Transferring Complete 1:Transferring *)
  NodeAddr : INT;  (* Executing Axis Number *)
  Error : BOOL;  (* Error *)
  ErrorID : WORD;  (* Error Code *)
END_VAR
VAR
  WAIT : BOOL;  (* First Cycle Wait Bit *)
  UnitSelect_Tmp : INT;  (* SCB/Select SCU Bit storage(internal variables) *)
  Type_W AT W0 : WORD;  (* Address type WR start address *)
  Type_Io AT 0 : WORD;  (* Address type IO start address *)
  Type_H AT H0 : WORD;  (* Address type HR start address *)
  Type_D AT D0 : WORD;  (* Address type DM start address *)
  Tmp_IR : ARRAY[0..3] OF DINT;  (* Temporary IR for internal variables *)
  Tmp_Data : ARRAY[0..30] OF WORD;  (* For internal Calculation *)
  Time_Value : UINT;  (* Interval Check Time Present Value *)
  Status_Inv_No : INT;  (* Status Command Slave Number *)
  Status_Commmnd_INT : BOOL;  (* Status Interrupt Flag *)
  Status_Commmnd_Enable : BOOL;  (* Enable Execution Status Command *)
  Status_2Cp : WORD;  (* second word of coils beginning with coil 1F to 2E *)
  Status_2C : WORD;  (* Register 2C Response Data *)
  Set_IR AT 0 : WORD;  (* Index register temporary setting *)
  Scanlist_Tmp : DWORD;  (* Scanlist storage *)
  SaveIR : ARRAY[0..3] OF DINT;  (* IR0toIR3 *)
  SaveDR : WORD;  (* DR0 *)
  Response_NG : BOOL;  (* Response error *)
  Response_Data : ARRAY[0..20] OF WORD;  (* CMND response data *)
  Response_CodeNG : BOOL;  (* Response end code error *)
  PortNo_Tmp : INT;  (* Serial port No. storage(internal variables) *)
  Phase : WORD;  (* Process Procedure *)
  P_FreeRunningCounter_10 AT A0 : UINT;  (* 10ms free running incremental counter *)
  P_Error : BOOL;  (* Error Flag *)
  P_EM_MaxNo AT A338 : INT;  (* EM bank size *)
  P_ComPort_WatchResTime AT A581 : INT;  (* FB Communications command response Monitor time *)
  P_ComPort_Retry AT A580 : WORD;  (* FB Communications command retry count *)
  P_ComPort_Finished0_7 AT A214 : WORD;  (* Communications Complete Cycle Bit *)
  P_ComPort_AutoAlloc_Available AT A202.15 : BOOL;  (* Auto allocation avarable bit *)
  P_ComPort_AllocatedNumber AT A218 : INT;  (* Network port No. *)
  Ok_WR : BOOL;  (* Selected WR area range OK *)
  Ok_IO : BOOL;  (* Selected CIO area range OK *)
  Ok_HR : BOOL;  (* Selected HR area range OK *)
  Ok_EM : BOOL;  (* Selected EM area range OK *)
  Ok_DM : BOOL;  (* Selected DM area range OK *)
  Ok_Bit : BOOL;  (* Range Check OK Bit *)
  Offset : DINT;  (* For Address Culcurate *)
  No : INT;  (* MatrixNo *)
  NG_Bit : BOOL;  (* Range Check NG Bit *)
  MSGAreaNo_Tmp : INT;  (* Message Area Number storage(internal variables) *)
  MSGAreaID_Tmp : WORD;  (* Message Area Classification storage(internal variables) *)
  ModelTypeMV_Tmp : DWORD;  (* MV/RVClassification storage(internal variables) *)
  Message_Command_Done : BOOL;  (* Exist Message Command Flag *)
  Last_Area_Status : ARRAY[0..61] OF WORD;  (* The Last Time IOM Status Condition *)
  Inv_Use_Count : INT;  (* Amount of Use Inverter Number *)
  Inv_Status_Count : INT;  (* Inverter Status Command Execution Number *)
  Inv_NodeArea : ARRAY[0..31] OF WORD;  (* Applicable Axis Inverter Model and Number Store Area *)
  INV_Error : BOOL;  (* Inverter Error *)
  Inv_Command_Change_Position : INT;  (* Inverter Write Command Changing Position *)
  IntervalCount_Tmp : UINT;  (* Interval storage(internal variables) *)
  IntervalCount_Compare : INT;  (* IntervalCompare Value *)
  Interval_TimeUp : BOOL;  (* Interval Time Up *)
  Interval_Start : BOOL;  (* Interval Count Start *)
  FreeRunningCounter_Tmp : UINT;  (* 10ms free running incremental counter record *)
  Error_Skip : BOOL;  (* Fatal Error Skip Flag *)
  EM_NoCheck : INT;  (* EM bank size check area *)
  EM_No_Tmp2 : UDINT;  (* EM area Calculation area 2 *)
  EM_No_Tmp1 : INT;  (* EM area Calculation area 1 *)
  Directive_Data : ARRAY[0..1] OF WORD;  (* Command data *)
  Data_Change : BOOL;  (* Detect input data change *)
  Control_Data : ARRAY[0..5] OF WORD;  (* CMND control data *)
  Command_Fin : BOOL;  (* CMND Transferring End *)
  Command_Data_Change2 : BOOL;
  Command_Data_Change : BOOL;  (* Write Command Data Changing *)
  Command_Data : ARRAY[0..21] OF WORD;  (* CMND command data *)
  Command_CheckNo : INT;  (* Write Command Check Complete Number *)
  CMNDPort : INT;  (* Port Number 1(Automatic Setting) *)
  BUSY_Run : BOOL;  (* Internal Processing Flag *)
  AreaNo_Tmp : INT;  (* Using Area Number storage(internal variables) *)
  AreaID_Tmp : WORD;  (* Using Area Classification storage(internal variables) *)
  AddressOk_Bit : BOOL;  (* Addrss Range Check OK Bit *)
  maxindex : UINT;  (* maximum possible inverters *)
  index : UINT;  (* index in the for next loop *)
  controlw : WORD;  (* controlword *)
  index2 : UINT;
  index3 : UINT;
  index4 : INT;  (* = index + 16 *)
  index5 : INT;  (* = index + 16 *)
  index6 : INT;  (* index3 +32 *)
  index7 : INT;
  Inv_Type_RX : BOOL;
END_VAR

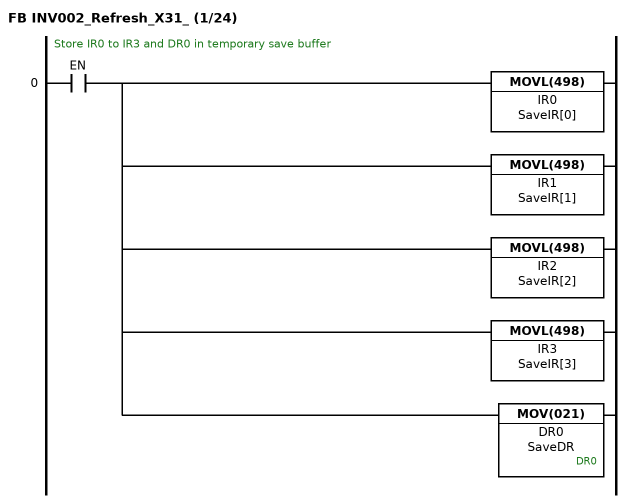
; rung 0: Store IR0 to IR3 and DR0 in temporary save buffer
LD EN
MOVL(498) IR0 SaveIR[0]
MOVL(498) IR1 SaveIR[1]
MOVL(498) IR2 SaveIR[2]
MOVL(498) IR3 SaveIR[3]
MOV(021) DR0 SaveDR  ; DR0

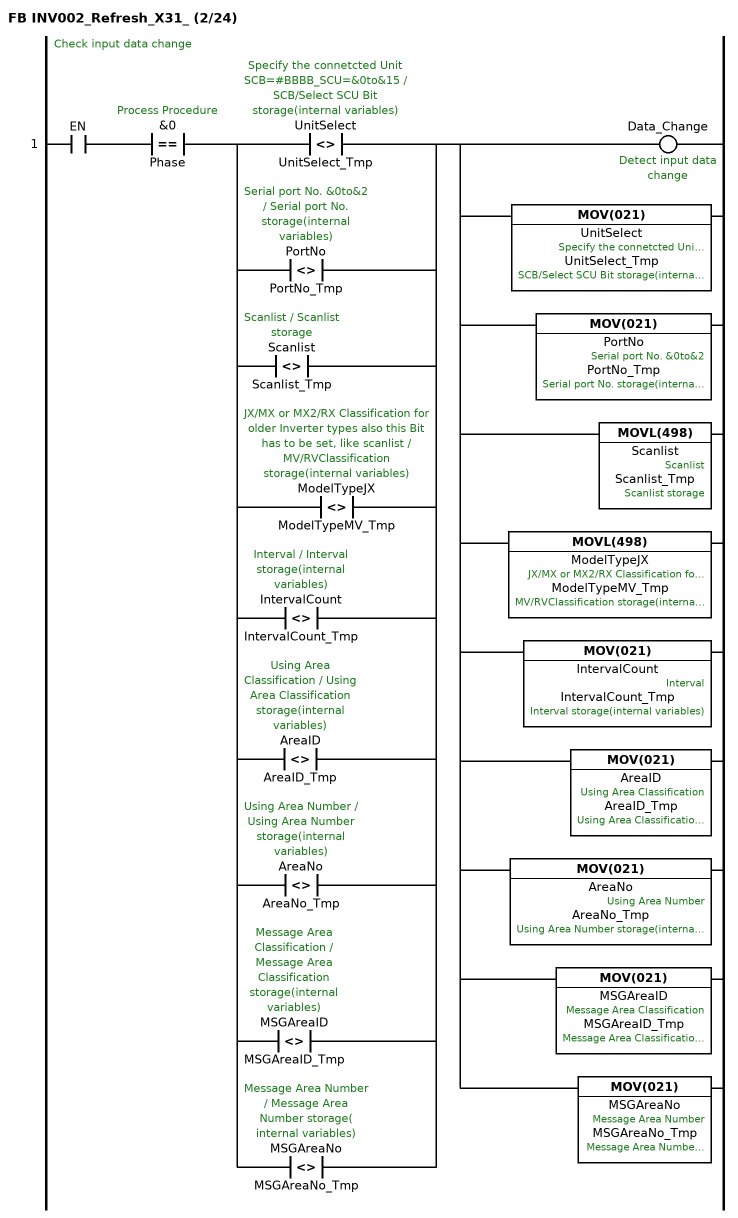
; rung 1: Check input data change
LD EN
AND=(300) &0 Phase  ; Process Procedure
LD<>(305) UnitSelect UnitSelect_Tmp  ; Specify the connetcted Unit SCB=#BBBB_SCU=&0to&15, SCB/Select SCU Bit storage(internal variables)
OR<>(305) PortNo PortNo_Tmp  ; Serial port No. &0to&2, Serial port No. storage(internal variables)
OR<>L(306) Scanlist Scanlist_Tmp  ; Scanlist, Scanlist storage
OR<>L(306) ModelTypeJX ModelTypeMV_Tmp  ; JX/MX or MX2/RX Classification for older Inverter types also this Bit has to be set, like scanlist, MV/RVClassification storage(internal variables)
OR<>(305) IntervalCount IntervalCount_Tmp  ; Interval, Interval storage(internal variables)
OR<>(305) AreaID AreaID_Tmp  ; Using Area Classification, Using Area Classification storage(internal variables)
OR<>(305) AreaNo AreaNo_Tmp  ; Using Area Number, Using Area Number storage(internal variables)
OR<>(305) MSGAreaID MSGAreaID_Tmp  ; Message Area Classification, Message Area Classification storage(internal variables)
OR<>(305) MSGAreaNo MSGAreaNo_Tmp  ; Message Area Number, Message Area Number storage(internal variables)
ANDLD
OUT Data_Change  ; Detect input data change
MOV(021) UnitSelect UnitSelect_Tmp  ; Specify the connetcted Unit SCB=#BBBB_SCU=&0to&15, SCB/Select SCU Bit storage(internal variables)
MOV(021) PortNo PortNo_Tmp  ; Serial port No. &0to&2, Serial port No. storage(internal variables)
MOVL(498) Scanlist Scanlist_Tmp  ; Scanlist, Scanlist storage
MOVL(498) ModelTypeJX ModelTypeMV_Tmp  ; JX/MX or MX2/RX Classification for older Inverter types also this Bit has to be set, like scanlist, MV/RVClassification storage(internal variables)
MOV(021) IntervalCount IntervalCount_Tmp  ; Interval, Interval storage(internal variables)
MOV(021) AreaID AreaID_Tmp  ; Using Area Classification, Using Area Classification storage(internal variables)
MOV(021) AreaNo AreaNo_Tmp  ; Using Area Number, Using Area Number storage(internal variables)
MOV(021) MSGAreaID MSGAreaID_Tmp  ; Message Area Classification, Message Area Classification storage(internal variables)
MOV(021) MSGAreaNo MSGAreaNo_Tmp  ; Message Area Number, Message Area Number storage(internal variables)

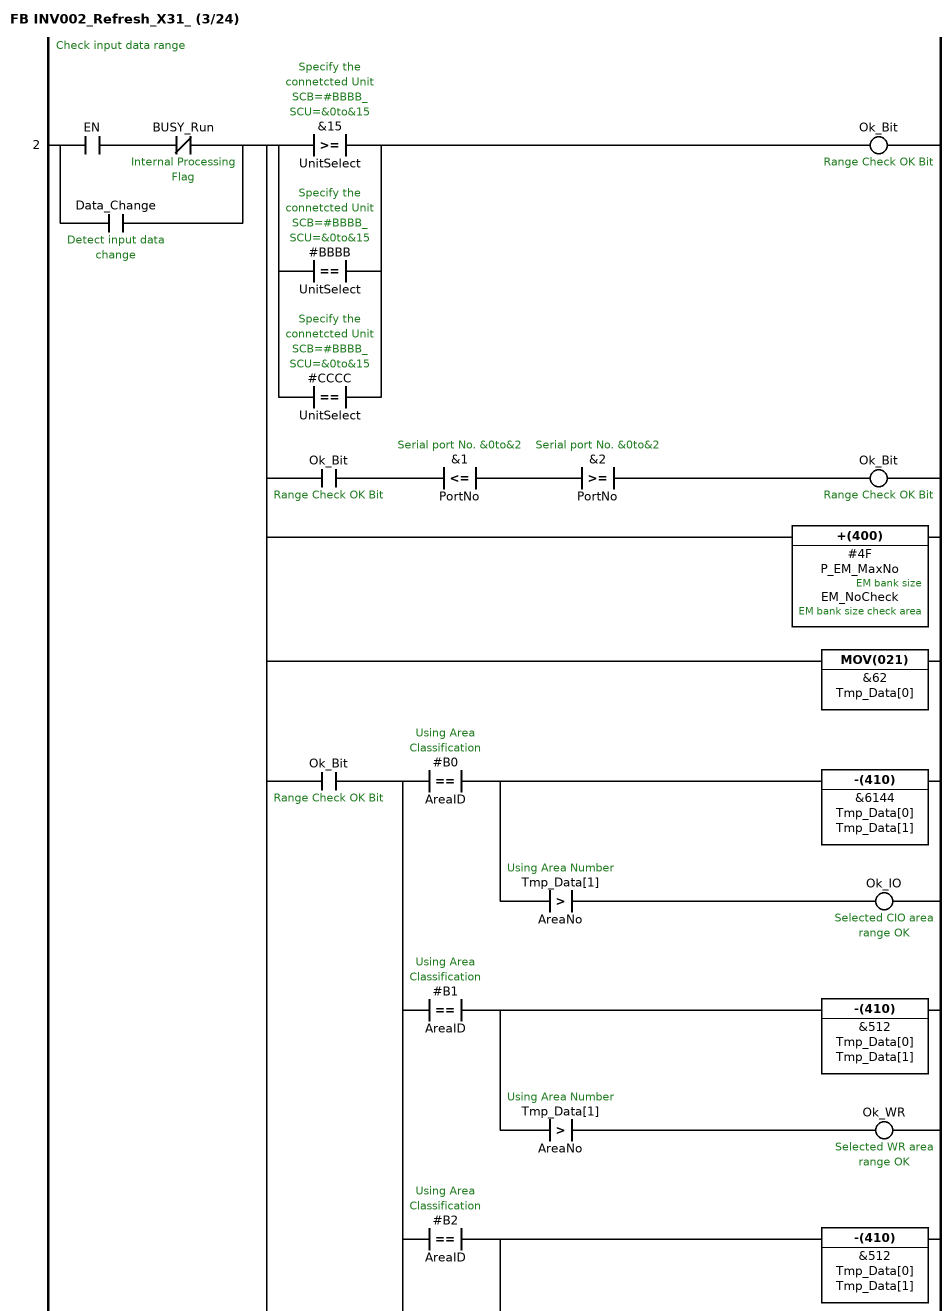

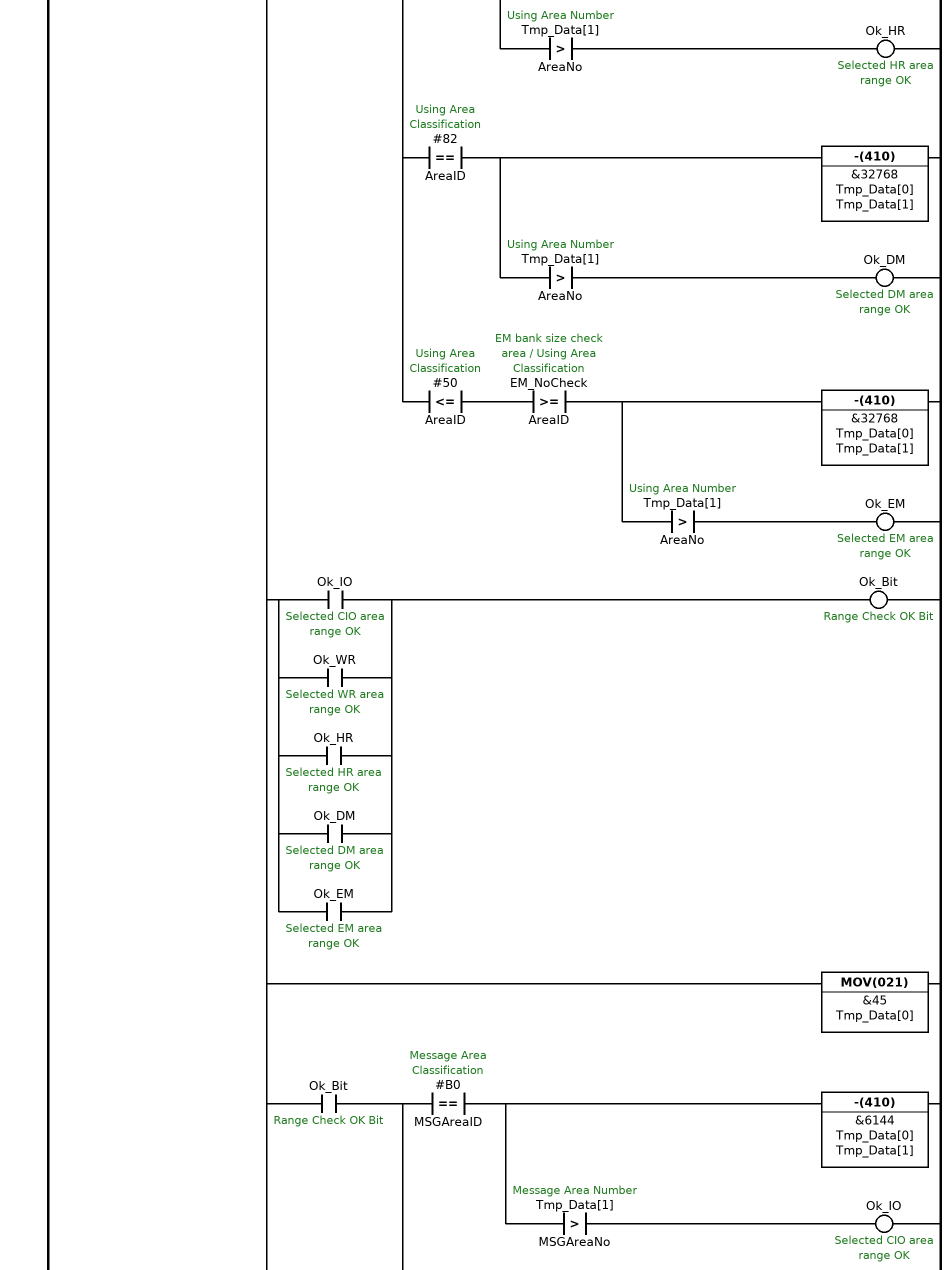

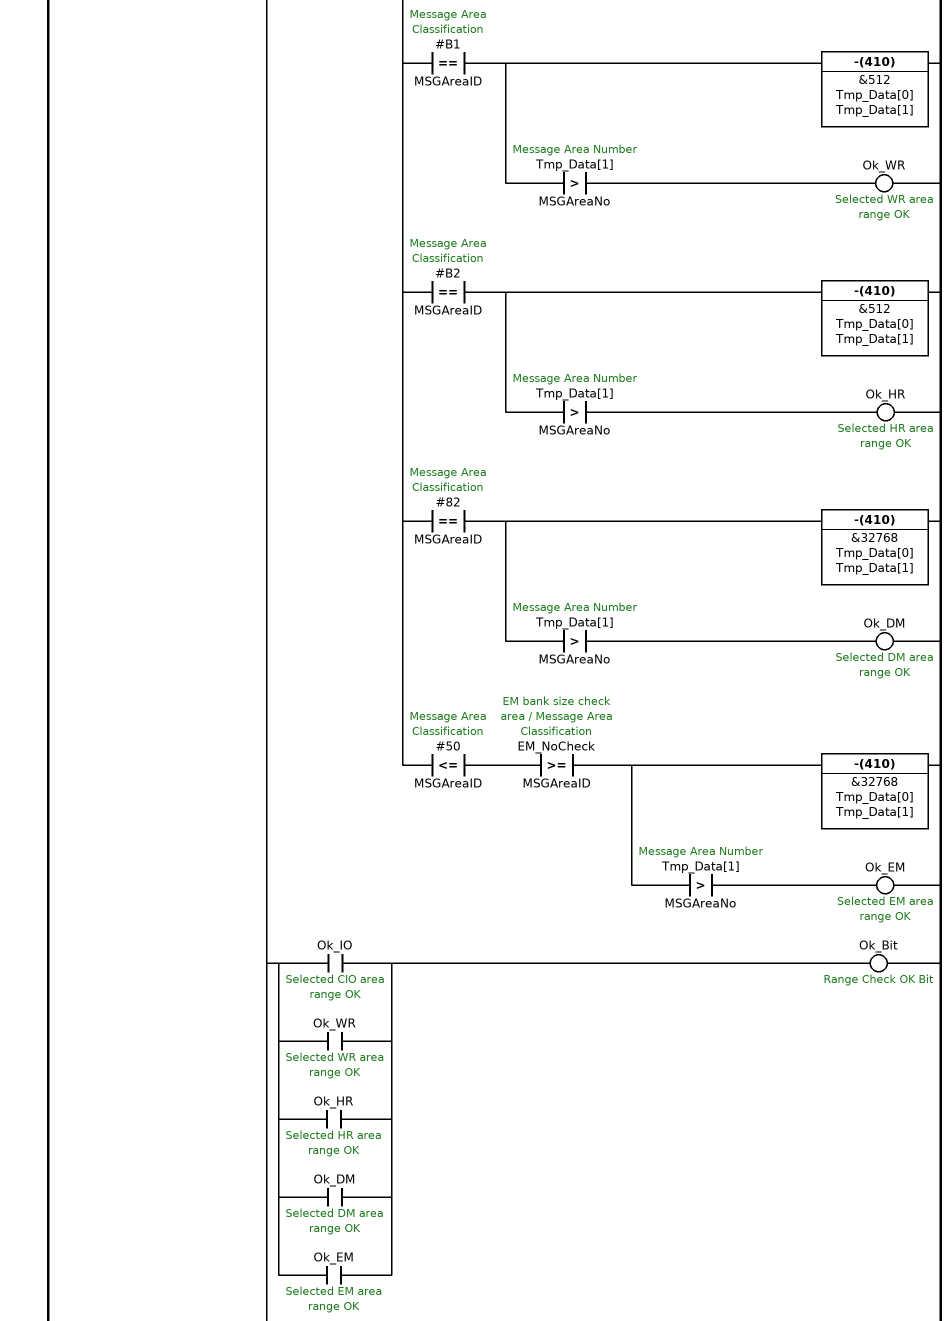

